(*			
	EVERDE sp. z o.o.
	Rafał Osajda		16.07.2025		TC 4024.66
	Lampka rozszerzona o moduł FB_Impuls co integruje w niej możlwiość mgania lub świecenie ciągłego
*)
FUNCTION_BLOCK FB_LampBlinking EXTENDS FB_Lamp IMPLEMENTS ITF_LampBlinking
VAR
	fbImpulse				: FB_BaseImpulse;
END_VAR

(*			
	EVERDE sp. z o.o.
	Rafał Osajda		05.02.2025		TC 4026.13		wer. 0.0.0.1
	Sterowanie swieceniem lampki - włącz/wyłącz
*)
METHOD Control
VAR_INPUT
	bIN	: BOOL;
END_VAR
IF (bIN) THEN
	THIS^.fbImpulse.SetExecuteOn ();
ELSE
	THIS^.fbImpulse.SetExecuteOff ();
END_IF
END_METHOD

(*			
	EVERDE sp. z o.o.
	Rafał Osajda		27.03.2025		TC 4024.66
	Wywolanie co cykl operacji 
*)
METHOD PUBLIC ExecuteEveryCycle_Operation
VAR_INPUT
END_VAR
SUPER^.ExecuteEveryCycle_Operation ();

THIS^.fbImpulse ();
END_METHOD

(*			
	EVERDE sp. z o.o.
	Rafał Osajda		27.03.2025		TC 4024.66
	Aktualizacja flag 
*)
METHOD PUBLIC ExecuteEveryCycle_Status
VAR_INST
END_VAR
SUPER^.ExecuteEveryCycle_Status ();

THIS^.bOut		:= THIS^.fbImpulse.GetExit ();
END_METHOD

(*			
	EVERDE sp. z o.o.
	Rafał Osajda		31.01.2025		TC 4026.13		wer. 0.0.0.1
	Sterowanie działem ipulsatora 
*)
METHOD PUBLIC SetBlink
VAR_INPUT
	bIN				: bool;
END_VAR
THIS^.fbImpulse.SetFlashing (bIN	:= bIN);
END_METHOD

(*			
	EVERDE sp. z o.o.
	Rafał Osajda		05.02.2025		TC 4026.13		wer. 0.0.0.1
	Wylacza lampke
*)
METHOD SetOff
THIS^.fbImpulse.SetExecuteOff ();
END_METHOD

(*			
	EVERDE sp. z o.o.
	Rafał Osajda		05.02.2025		TC 4026.13		wer. 0.0.0.1
	Wlacza lampke - praca ciągła
*)
METHOD SetOn
THIS^.fbImpulse.SetExecuteOn ();
END_METHOD

METHOD PUBLIC SetShine
VAR_INPUT
	bIN				: BOOL;
END_VAR
IF (bIN) THEN
	THIS^.fbImpulse.SetExecuteOn ();
ELSE
	THIS^.fbImpulse.SetExecuteOff ();
END_IF
END_METHOD

(*			
	EVERDE sp. z o.o.
	Rafał Osajda		31.01.2025		TC 4026.13		wer. 0.0.0.1
	Ustawia czas zgaszonej lampki
*)
METHOD PUBLIC SetTimeOff
VAR_INPUT
	rIN					: REAL;
END_VAR
THIS^.fbImpulse.SetTimeOff (rIN	:= rIN);
END_METHOD

(*			
	EVERDE sp. z o.o.
	Rafał Osajda		31.01.2025		TC 4026.13		wer. 0.0.0.1
	
*)
METHOD PUBLIC SetTimeOn
VAR_INPUT
	rIN						: REAL;
END_VAR
THIS^.fbImpulse.SetTimeOn (rIN	:= rIN);
END_METHOD

METHOD PUBLIC SetWork
VAR_INPUT
	bShine		: BOOL;
	bBlink		: BOOL;
	rTimeOn		: REAL;
	rTimeOff	: REAL;
END_VAR
THIS^.fbImpulse.SetTimeOn (rIN := rTimeOn);
THIS^.fbImpulse.SetTimeOff (rIN := rTimeOff);
THIS^.SetShine (bIN	:= bShine);
THIS^.SetBlink (bIN := bBlink);
END_METHOD

END_FUNCTION_BLOCK

(* stored: Version 1.1.0.1
   POU FB_LampBlinking: Id {dcff81a1-6dd7-4eaf-907a-2248d98a1fd0}, SpecialFunc None
   Folder Impuls: Id {00302c85-f7fe-4010-b913-cb28ac209e80}
   Folder Lampka: Id {1ce39044-512f-4976-97b5-7f5d1cfcc4ca}
   Method Control: Id {89cae73f-2289-0458-1edf-fb704988ff0f}
   Method ExecuteEveryCycle_Operation: Id {3122b5f5-fb1e-4355-b29b-0ca3046f4573}
   Method ExecuteEveryCycle_Status: Id {22023be3-3f2d-479c-beea-467a1af9fb42}
   Method SetBlink: Id {7308fc6d-0df1-0fc9-3448-90bfe4f60c6d}
   Method SetOff: Id {74da1db2-cae1-4989-b15d-2e841810dcc3}
   Method SetOn: Id {3cba340c-0e1a-4db9-b5dc-78c607c4f1e1}
   Method SetShine: Id {d73aa7c8-66fb-44b9-abcb-6defbf850207}
   Method SetTimeOff: Id {6e8b987e-d352-044d-0d8b-d018d73edb47}
   Method SetTimeOn: Id {6984913b-06ff-0018-00ab-a77455e9d2b1}
   Method SetWork: Id {394fd72e-1ef7-4d61-b407-9f1d7f9d1d0d} *)
